FUNCTION FC_6strConcat : T_DEFAULT_STR		// Concatenates 4 strings
VAR_INPUT
	iStr1:		T_DEFAULT_STR;
	iStr2:		T_DEFAULT_STR;
	iStr3:		T_DEFAULT_STR;
	iStr4:		T_DEFAULT_STR;
	iStr5:		T_DEFAULT_STR;
	iStr6:		T_DEFAULT_STR;
END_VAR

FC_6strConcat := CONCAT(FC_5strConcat(iStr1, iStr2, iStr3, iStr4, iStr5), iStr6);

END_FUNCTION

(* stored: Version 1.1.0.1, ProductVersion 3.1.4026.18
   POU FC_6strConcat: Id {96264cbe-6f80-4c4e-a33f-b91da96fab0f}, SpecialFunc None *)
